FUNCTION_BLOCK FB_EL3356_0010
VAR_INPUT

	i_tInputFreeze				:TIME:=T#50MS;
	i_rInputFreezeTreshold		:REAL:=10;
END_VAR
VAR_OUTPUT
		(* Status Flag*)
	o_obUnderrange				:BOOL;		//低於範圍
	o_bOverrange				:BOOL;		//超出範圍 
	o_bDataInvalid				:BOOL;		//資料無效 
	o_bError					:BOOL;		//Error
	o_bCalibrationInProgress	:BOOL;		//
	o_bSteadyState				:BOOL;		//穩定中 
	o_bTxPDOToggle				:BOOL;		//刷新資料
	o_bSyncError				:BOOL;		//
	o_rWeight					:REAL;
	strStatus					:STRING(100);
	strSampleMode				:STRING(100);			
END_VAR
VAR
	(* process data OUT*)
	wControl AT %Q*:WORD;
	(* process data IN*)
	wStatus AT %I*:WORD;
	rValue_REAL AT %I*:REAL;
	nValue_Supply AT %I*:DINT;		(*only for voltage measurement, change PDO settings"*)
	nValue_Bridge AT %I*:DINT;		(*only for voltage measurement, change PDO settings"*)
	stEcSlaveAmsNetAdr AT %I*:ST_AmsAddr;
	bWcState AT %I*:BOOL;
	wState AT %I*:WORD;

	
		(* Control commands *)
	bStartManualCalib	:BOOL;		//開始校準	-Control 
	bDisableCalibration	:BOOL;		//停止校準	-Control
	bSampleMode			:BOOL;		//sampleMode	-Control
	bTara				:BOOL;		//去皮		-Control
	//////////
	sEcSlaveAmsNetAdr:T_AmsNetId;
	rValue:REAL;

	fbCoE		:ARRAY [0..10] OF  FB_EcCoESdoWrite;
	wCoeData	:WORD;
	dwCoeData	:DWORD;
	bTermError:BOOL;
	nCntCalibrations:UDINT;
	sfCalibInProgress:R_TRIG;

	_bInitial		,_bSetLoadcell,_bSetRefLoad,_bSetScaleFactor,_bSetZeroCali,_bSetLoadCali ,_bSetCommand,_bTara		:BOOL;
	_Initialbuff	,_SetLoadcell,_SetRefLoad	,_SetScaleFactor,_SetZeroCali,_SetLoadCali	,_SetCommand,_Tara		:WORD;
	

	rValueDiff, rValueL:REAL;
	bActivateAutoInputFreeze:BOOL;
	tofInputFreeze:TOF;
	tInputFreeze:TIME:=T#50MS;
	tTara	:TON := (PT := TIME#500ms);
	sfCntInputFreeze:R_TRIG;
	nCntInputFreeze:UDINT;


END_VAR

	(*example program for EL3356(-0010)
	this demo is designed only for load cell connection, not for 2channel voltage measurement*)

	(*get terminal information*)
o_bOverrange := wStatus.1;
o_bDataInvalid := wStatus.3;
o_bError := wStatus.6;
o_bCalibrationInProgress := wStatus.7;
o_bSteadyState := wStatus.8;
o_bSyncError := wStatus.13;
o_bTxPDOToggle := wStatus.15;
	(*triggers*)
	
//sfZeroCalibration(CLK:=i_bCmd_ZeroCalibration);
//sfFullCalibration(CLK:=i_bCmd_FullCalibration);
//sfTara(CLK:=i_bCmd_Tara);
//sfTaraEEProm(CLK:=i_bCmd_TaraEEProm);
//sfInitial(CLK:= i_bInitial);
//sfWriteLoadcellMaxWeight(CLK:= i_bWriteLoadcellMaxWeight);
//sfbWriteRefWeight(CLK:= i_bWriteRefWeight);


	(*value: Integer or Real value*)
IF (rValue_REAL <> 0) THEN	(*select currently used input data*)
	rValue := rValue_REAL;
	rValue := 0;
END_IF

	(*status*)
IF bWcState THEN
	strStatus := 'Wc fail';
	bTermError := TRUE;
ELSIF NOT (wState.3) THEN
	strStatus := 'Slave not in OP';
	bTermError := TRUE;
ELSIF o_bDataInvalid THEN
	strStatus := 'DataInvalid';
	bTermError := TRUE;
ELSIF o_bError THEN
	strStatus := 'Channel Error';
	bTermError := TRUE;
ELSIF o_bOverrange THEN
	strStatus := 'Overrange';
	bTermError := TRUE;
ELSE
	strStatus := 'ok';
	bTermError := FALSE;
END_IF

	(*sample mode 0/1*)
strSampleMode := SEL(bSampleMode, '0', '1');

	(*count calibrations*)
sfCalibInProgress(CLK:= o_bCalibrationInProgress, Q=> );
nCntCalibrations := SEL(sfCalibInProgress.Q , nCntCalibrations, nCntCalibrations+ 1);

	(*Coe parameter administration*)
sEcSlaveAmsNetAdr := F_CreateAmsNetId(nIds:=stEcSlaveAmsNetAdr.netId );

	(*test input freeze
this lines are for a small demonstration of Input freeze: when difference of loadvalue, compared to last PLC cycle, is over rInputFreezeTreshold
then InputFreeze is activated by tofInputFreeze for some time. See screenshot in documentation for further explanations*)
rValueDiff := rValue - rValueL;
rValueL := rValue;
tofInputFreeze(IN:= bActivateAutoInputFreeze AND (ABS(rValueDiff) >i_rInputFreezeTreshold) , PT:= tInputFreeze, Q=> , ET=> );
sfCntInputFreeze(CLK:= tofInputFreeze.Q , Q=> );
nCntInputFreeze := SEL(sfCntInputFreeze.Q , nCntInputFreeze, nCntInputFreeze+ 1);

(*++++++++++++++ CoE communication ++++++++++++++++++++++*)
IF NOT _bInitial THEN
	fbCoE[0](bExecute 	:= FALSE);
	_Initialbuff	:= 0;
END_IF
_bInitial:= FALSE;
//
IF NOT _bSetLoadcell THEN
	fbCoE[1](bExecute 	:= FALSE);
	_SetLoadcell	:= 0;
END_IF
_bSetLoadcell:=FALSE;
//
IF NOT _bSetRefLoad THEN
	fbCoE[2](bExecute 	:= FALSE);
	_SetRefLoad	:= 0;
END_IF
_bSetRefLoad:=FALSE;
//
IF NOT _bSetScaleFactor THEN
	fbCoE[3](bExecute 	:= FALSE);
	_SetScaleFactor	:= 0;
END_IF
_bSetScaleFactor:= FALSE;

//
IF NOT _bSetZeroCali THEN
	fbCoE[4](bExecute 	:= FALSE);
	_SetZeroCali	:= 0;
END_IF
_bSetZeroCali	:= FALSE;
//
IF NOT _bSetLoadCali THEN
	fbCoE[5](bExecute 	:= FALSE);
	_SetLoadCali	:= 0;
END_IF
_bSetLoadCali	:= FALSE;
//
IF NOT _bSetCommand THEN
	fbCoE[6](bExecute 	:= FALSE);
	_SetCommand	:= 0;
END_IF
_bSetCommand	:= FALSE;

//
IF NOT _bTara THEN
	tTara(IN:=FALSE);
	_Tara	:= 0;
	bTara	:= FALSE;
END_IF
_bTara:=FALSE;
	(*output data to terminal*)
wControl.0 := bStartManualCalib;
wControl.1 := bDisableCalibration;
//wControl.2 := i_bInputFreeze OR tofInputFreeze.Q ;
wControl.3 := bSampleMode;
wControl.4 := bTara;

o_rWeight:= rValue_REAL;
//Ext

METHOD GetTara : BOOL
VAR_INPUT
END_VAR
_bTara	:= TRUE;

CASE _Tara OF
	0: 
		bTara	:= TRUE;
		tTara(IN:= TRUE);
		IF tTara.Q THEN
			tTara(IN:= FALSE);
			_Tara	:= 5;
		END_IF

	5:
		GetTara:= TRUE;
END_CASE
END_METHOD

METHOD Initialization : BOOL
VAR_INPUT
END_VAR
//修改CoE object 0x1011:01值为1684107116恢复出厂设置
_bInitial	:= TRUE;

CASE _Initialbuff OF
	0:
		dwCoeData := 1684107116; (* Command zerocalibration*)
		fbCoE[0](
			sNetId		:= sEcSlaveAmsNetAdr,
			nSlaveAddr 	:= stEcSlaveAmsNetAdr.port,
			nSubIndex 	:= 16#01,
			nIndex 		:= 16#1011,
			pSrcBuf 	:= ADR(dwCoeData),
			cbBufLen 	:= SIZEOF(dwCoeData),
			bExecute 	:= TRUE,
			tTimeout 	:= T#5S		
			);
		IF fbCoE[0].bBusy THEN
			_Initialbuff	:= 1;
		END_IF;
			
	1:
		fbCoE[0]();				
		IF NOT fbCoE[0].bBusy THEN
			_Initialbuff	:= 2;
			IF fbCoE[0].bError THEN
				_Initialbuff	:= 5;
			END_IF
		END_IF;	
	2:
		Initialization		:= TRUE;
		fbCoE[0](bExecute 	:= FALSE);
	5:
		Initialization		:= TRUE;
		fbCoE[0](bExecute 	:= FALSE);		
END_CASE
END_METHOD

METHOD SetLoadCalibration : BOOL
VAR_INPUT
END_VAR
_bSetLoadCali	:= TRUE;

CASE _SetLoadCali OF
	0:
		_SetLoadCali	:= 1;
	
	1:
		wCoeData	:= 16#0102;
		fbCoE[5](
			sNetId		:= sEcSlaveAmsNetAdr,
			nSlaveAddr 	:= stEcSlaveAmsNetAdr.port,
			nSubIndex 	:= 16#01,
			nIndex 		:= 16#FB00,
			pSrcBuf 	:= ADR(wCoeData),
			cbBufLen 	:= SIZEOF(wCoeData),
			bExecute 	:= TRUE,
			tTimeout 	:= T#5S		
			);
		IF fbCoE[5].bBusy THEN
			_SetLoadCali	:=2;
		END_IF;
			
	2:
		fbCoE[5]();				
		IF NOT fbCoE[5].bBusy THEN
			_SetLoadCali	:= 3;
			IF fbCoE[5].bError THEN
				_SetLoadCali	:= 5;
			END_IF
		END_IF;	
	3:
		SetLoadCalibration		:= TRUE;
		fbCoE[5](bExecute 	:= FALSE);
	5:

		fbCoE[5](bExecute 	:= FALSE);		
END_CASE
END_METHOD

METHOD SetNomialLoad : BOOL
VAR_INPUT
	MaxWeight:REAL;
END_VAR
//8.	0x8000:24 ("额定值") ，本例的传感器为最大称重1kg，那么就输入1000 
_bSetLoadcell	:= TRUE;

CASE _SetLoadcell OF
	0:
		IF MaxWeight = 0.0 THEN
			_SetLoadcell	:=5;
			ELSE
			_SetLoadcell	:= 1;
		END_IF
	1:
		fbCoE[1](
			sNetId		:= sEcSlaveAmsNetAdr,
			nSlaveAddr 	:= stEcSlaveAmsNetAdr.port,
			nSubIndex 	:= 16#24,
			nIndex 		:= 16#8000,
			pSrcBuf 	:= ADR(MaxWeight),
			cbBufLen 	:= SIZEOF(MaxWeight),
			bExecute 	:= TRUE,
			tTimeout 	:= T#5S		
			);
		IF fbCoE[1].bBusy THEN
			_SetLoadcell	:=2;
		END_IF;
			
	2:
		fbCoE[1]();				
		IF NOT fbCoE[1].bBusy THEN
			_SetLoadcell	:= 3;
			IF fbCoE[1].bError THEN
				_SetLoadcell	:= 5;
			END_IF
		END_IF;	
	3:
		SetNomialLoad		:= TRUE;
		fbCoE[1](bExecute 	:= FALSE);
	5:

		fbCoE[1](bExecute 	:= FALSE);		
END_CASE
END_METHOD

METHOD SetRefLoad : BOOL
VAR_INPUT
	RefLoad:REAL;
END_VAR
//500g的砝码在 0x8000:28 校准负载填写500, (0x8000:24)额定负载填写1000。

_bSetRefLoad	:= TRUE;

CASE _SetRefLoad OF
	0:
		IF RefLoad = 0.0 THEN
			_SetRefLoad	:=5;
			ELSE
			_SetRefLoad	:= 1;
		END_IF
	1:
		fbCoE[2](
			sNetId		:= sEcSlaveAmsNetAdr,
			nSlaveAddr 	:= stEcSlaveAmsNetAdr.port,
			nSubIndex 	:= 16#28,
			nIndex 		:= 16#8000,
			pSrcBuf 	:= ADR(RefLoad),
			cbBufLen 	:= SIZEOF(RefLoad),
			bExecute 	:= TRUE,
			tTimeout 	:= T#5S		
			);
		IF fbCoE[2].bBusy THEN
			_SetRefLoad	:=2;
		END_IF;
			
	2:
		fbCoE[2]();				
		IF NOT fbCoE[2].bBusy THEN
			_SetRefLoad	:= 3;
			IF fbCoE[2].bError THEN
				_SetRefLoad	:= 5;
			END_IF
		END_IF;	
	3:
		SetRefLoad		:= TRUE;
		fbCoE[2](bExecute 	:= FALSE);
	5:

		fbCoE[2](bExecute 	:= FALSE);		
END_CASE
END_METHOD

METHOD SetScaleFactor : BOOL
VAR_INPUT
	ScaleFactor	:REAL;
END_VAR
//0x8000:27 校准负载填写1單位kg , 1000/g

_bSetScaleFactor	:= TRUE;

CASE _SetScaleFactor OF
	0:
		IF ScaleFactor = 0.0 THEN
			_SetScaleFactor	:=5;
			ELSE
			_SetScaleFactor	:= 1;
		END_IF
	1:
		fbCoE[3](
			sNetId		:= sEcSlaveAmsNetAdr,
			nSlaveAddr 	:= stEcSlaveAmsNetAdr.port,
			nSubIndex 	:= 16#27,
			nIndex 		:= 16#8000,
			pSrcBuf 	:= ADR(ScaleFactor),
			cbBufLen 	:= SIZEOF(ScaleFactor),
			bExecute 	:= TRUE,
			tTimeout 	:= T#5S		
			);
		IF fbCoE[3].bBusy THEN
			_SetScaleFactor	:=2;
		END_IF;
			
	2:
		fbCoE[3]();				
		IF NOT fbCoE[3].bBusy THEN
			_SetScaleFactor	:= 3;
			IF fbCoE[3].bError THEN
				_SetScaleFactor	:= 5;
			END_IF
		END_IF;	
	3:
		SetScaleFactor		:= TRUE;
		fbCoE[3](bExecute 	:= FALSE);
	5:

		fbCoE[3](bExecute 	:= FALSE);		
END_CASE
END_METHOD

METHOD SetZeroCalibration : BOOL
VAR_INPUT
END_VAR
_bSetZeroCali	:= TRUE;

//0x8000:27 校准负载填写1單位kg , 1000/g

CASE _SetZeroCali OF
	0:
		_SetZeroCali	:= 1;
	
	1:
		wCoeData	:= 16#0101;
		fbCoE[4](
			sNetId		:= sEcSlaveAmsNetAdr,
			nSlaveAddr 	:= stEcSlaveAmsNetAdr.port,
			nSubIndex 	:= 16#01,
			nIndex 		:= 16#FB00,
			pSrcBuf 	:= ADR(wCoeData),
			cbBufLen 	:= SIZEOF(wCoeData),
			bExecute 	:= TRUE,
			tTimeout 	:= T#5S		
			);
		IF fbCoE[4].bBusy THEN
			_SetZeroCali	:=2;
		END_IF;
			
	2:
		fbCoE[4]();				
		IF NOT fbCoE[4].bBusy THEN
			_SetZeroCali	:= 3;
			IF fbCoE[4].bError THEN
				_SetZeroCali	:= 5;
			END_IF
		END_IF;	
	3:
		SetZeroCalibration		:= TRUE;
		fbCoE[4](bExecute 	:= FALSE);
	5:

		fbCoE[4](bExecute 	:= FALSE);		
END_CASE
END_METHOD

METHOD WriteCommand : BOOL
VAR_INPUT
	wInputData	:WORD;
END_VAR
_bSetCommand	:= TRUE;

CASE _SetCommand OF
	0:
		_SetCommand	:= 1;
	
	1:
		wCoeData	:= wInputData;
		fbCoE[6](
			sNetId		:= sEcSlaveAmsNetAdr,
			nSlaveAddr 	:= stEcSlaveAmsNetAdr.port,
			nSubIndex 	:= 16#01,
			nIndex 		:= 16#FB00,
			pSrcBuf 	:= ADR(wCoeData),
			cbBufLen 	:= SIZEOF(wCoeData),
			bExecute 	:= TRUE,
			tTimeout 	:= T#5S		
			);
		IF fbCoE[6].bBusy THEN
			_SetCommand	:=2;
		END_IF;
			
	2:
		fbCoE[6]();				
		IF NOT fbCoE[6].bBusy THEN
			_SetCommand	:= 3;
			IF fbCoE[6].bError THEN
				_SetCommand	:= 5;
			END_IF
		END_IF;	
	3:
		WriteCommand		:= TRUE;
		fbCoE[6](bExecute 	:= FALSE);
	5:

		fbCoE[6](bExecute 	:= FALSE);		
END_CASE
END_METHOD

END_FUNCTION_BLOCK

(* stored: Version 1.1.0.1, ProductVersion 3.1.4024.16
   POU FB_EL3356_0010: Id {d7d7f3d2-0059-44e1-85f5-0272e0da6cbb}, SpecialFunc None
   Method GetTara: Id {067ff3c3-cba2-4eea-bfed-74a522ab6da2}
   Method Initialization: Id {bd1ce88e-9c1e-42b5-94ed-d0c5df17859c}
   Method SetLoadCalibration: Id {d4388e7f-93f1-497d-9c2b-7848ef4cf875}
   Method SetNomialLoad: Id {cd943a8c-5225-46dc-a54a-c851e9f1db26}
   Method SetRefLoad: Id {2ed8e764-7915-439e-917f-5713e4eaca38}
   Method SetScaleFactor: Id {7818337d-15dd-462e-ad88-007a15a7b932}
   Method SetZeroCalibration: Id {051e7a1d-1421-4657-bbb4-d93b6dd0d6b3}
   Method WriteCommand: Id {6552a2f7-073d-4a84-b097-b93e8d65a96a} *)
